(* IEC 61131-3 sources: PIDControlBackUpFolder/PIDControl, 3 files *)

(* ---- IDDone.st ---- *)
FUNCTION_BLOCK IDDone
	IF DoneIn = TRUE OR DoneOnce > 0 THEN
		Done := TRUE;
		DoneOnce := 1;
	ELSE
		Done := FALSE;
	END_IF
END_FUNCTION_BLOCK

(* ---- LocalFunctions.fun ---- *)
FUNCTION_BLOCK IDDone
	VAR_INPUT
		DoneIn : BOOL;
	END_VAR
	VAR_OUTPUT
		Done : BOOL;
	END_VAR
	VAR_IN_OUT
		DoneOnce : INT;
	END_VAR
END_FUNCTION_BLOCK

(* ---- Init.st ---- *)
PROGRAM _INIT

	AxisParameters.Position := 0.0;
	AxisParameters.Velocity := 10.0;
	AxisParameters.Acceleration := 50.0;
	AxisParameters.Deceleration := 50.0;

END_PROGRAM
